// SIMATIC S7-200 SMART project (STEP 7-Micro/WIN SMART), CPU SR40

SYMBOL_TABLE 表格 1
过程变量             VW0
PID输出            VW2
手动输入             VD4
给定值              VD8
YLAST1           VD100
YLAST2           VD104
YLAST3           VD108
END_SYMBOL_TABLE

SYMBOL_TABLE 系统符号
Always_On        SM0.0    // 始终接通
First_Scan_On    SM0.1    // 仅在第一个扫描周期时接通
Time_1_Intrvl    SMB35    // 指定中断 1 的时间间隔（从 1 - 255，以 1 ms 递增）。
END_SYMBOL_TABLE

ORGANIZATION_BLOCK MAIN:OB1
TITLE=程序注释
BEGIN
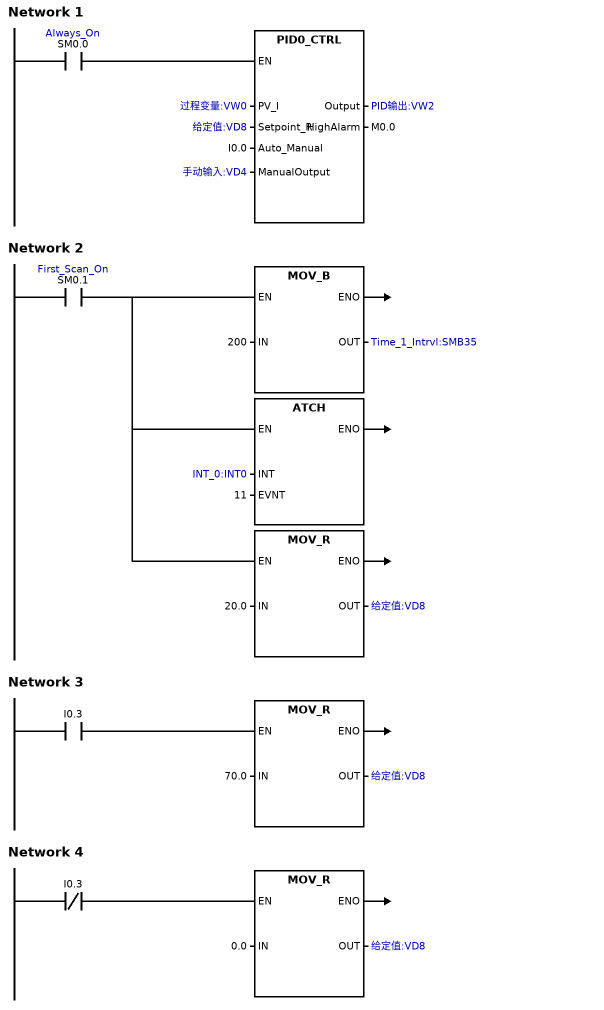
Network 1
// (network saved uncompiled; LAD cells follow)
// row 0: c0 -| |- Always_On:SM0.0  c1 --  c2 [PID0_CTRL EN:=power@row0, PV_I:=过程变量:VW0, Setpoint_R:=给定值:VD8, Auto_Manual:=I0.0, ManualOutput:=手动输入:VD4, Output=>PID输出:VW2, HighAlarm=>M0.0]
// row 1: c2 [box]
// row 2: c2 [box]
Network 2
LD     First_Scan_On:SM0.1
MOVB   200, Time_1_Intrvl:SMB35
ATCH   INT_0:INT0, 11
MOVR   20.0, 给定值:VD8
Network 3
LD     I0.3
MOVR   70.0, 给定值:VD8
Network 4
LDN    I0.3
MOVR   0.0, 给定值:VD8
END_ORGANIZATION_BLOCK

// SBR0: protected block, not included

// SBR1: protected block, not included

INTERRUPT_BLOCK INT_0:INT0
TITLE=中断例程注释
BEGIN
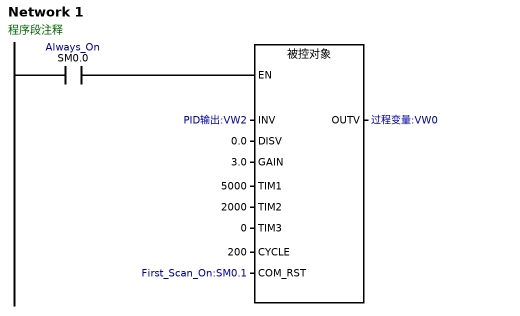
Network 1
// 程序段注释
LD     Always_On:SM0.0
CALL   被控对象:SBR0, PID输出:VW2, 0.0, 3.0, 5000, 2000, 0, 200, First_Scan_On:SM0.1, 过程变量:VW0
END_INTERRUPT_BLOCK

// INT1: protected block, not included
